{attribute 'linkalways'} 
{attribute 'no_explicit_call' := 'This FB is a CLASS and must be accessed using methods or properties'}
{attribute 'enable_dynamic_creation'}
FUNCTION_BLOCK Node_F_VN_MaxElementElementwise_UDINT EXTENDS VisionNode
VAR
    ipContainer : _ITcVnContainer;
    nMax : _UDINT(0);
    hrPrev : _HRESULT(S_OK);
    hresult : _HRESULT(S_OK);
END_VAR

METHOD PUBLIC  Clone : I_Node
VAR
	pNode : POINTER TO Node_F_VN_MaxElementElementwise_UDINT;
END_VAR
pNode := __NEW(Node_F_VN_MaxElementElementwise_UDINT);
Clone := pNode^;
END_METHOD

METHOD FB_init : BOOL
VAR_INPUT
	bInitRetains : BOOL; // if TRUE, the retain variables are initialized (warm start / cold start)
	bInCopyCode : BOOL;  // if TRUE, the instance afterwards gets moved into the copy code (online change)
END_VAR
AddInput('ipContainer', ipContainer);
AddInput('hrPrev', hrPrev);
AddOutput('ipContainer', ipContainer);
AddOutput('nMax', nMax);
AddOutput('hresult',hresult);
END_METHOD

METHOD PROTECTED OnExecute
hresult.Value := F_VN_MaxElementElementwise_UDINT(
    ipContainer := ipContainer.Value,
    nMax := nMax.Value,
    hrPrev:= hrPrev.Value);
END_METHOD

METHOD PUBLIC PreExecutionCheck
VAR_INPUT
	Check : I_PreExecutionChecks;
END_VAR
Check.IsTrue(ipContainer.IsValid, 'ipContainer must be a valid container');
Check.IsTrue(ipContainer.IsType(TC_GLOBAL_CONST_LIST.ContainerType_Vector_UDINT), 'ipContainer contains incorrect type');
END_METHOD

END_FUNCTION_BLOCK

(* stored: Version 1.1.0.1, ProductVersion 3.1.4026.13
   POU Node_F_VN_MaxElementElementwise_UDINT: Id {7d65dc49-1a33-4972-9efd-73c7ec916712}, SpecialFunc None
   Folder Constructor: Id {f49cedc7-dce4-4a23-a651-d72f921e5dc0}
   Method Clone: Id {3d6e815e-48b0-4544-8a3d-d9297b0f1ee2}
   Method FB_init: Id {4cfc90b8-b8eb-48d4-8d2b-bcfc686a3f3a}
   Method OnExecute: Id {261b4b72-b44b-4d74-8cd4-a5edf4017a0b}
   Method PreExecutionCheck: Id {c4c37f25-9583-4ffb-b362-c4f8bf0bedca} *)
